INTERFACE I_ENGINE_VALVE EXTENDS I_GENERAL_OBJECT

METHOD M_Close : BOOL
VAR_INPUT
END_VAR
END_METHOD

METHOD M_Open : BOOL
VAR_INPUT
END_VAR
END_METHOD

METHOD M_SetReady : BOOL
VAR_INPUT
END_VAR
END_METHOD

PROPERTY P_Closed : BOOL
GET
END_GET
END_PROPERTY

PROPERTY P_Open : BOOL
GET
END_GET
END_PROPERTY

PROPERTY P_ReadyState : BOOL
GET
END_GET
END_PROPERTY

PROPERTY P_Undefined : BOOL
GET
END_GET
END_PROPERTY

END_INTERFACE

(* stored: Version 1.1.0.1, ProductVersion 3.1.4024.12
   Itf I_ENGINE_VALVE: Id {7e3ceb72-8a0a-4c5a-9e38-262f19a4f12a}
   Method M_Close: Id {2ea4d968-aa32-49e9-92a5-3cfde55592cc}
   Method M_Open: Id {9b168fe1-6505-4f60-9e5c-4242991cd250}
   Method M_SetReady: Id {fdd3cae0-8774-4296-b5ba-55d8bd97d36c}
   Property P_Closed: Id {ff5951e8-0f3a-4262-bf83-1327a1158ec9}
   Get Get: Id {1a09b6d8-8ccb-4b68-ba38-3ee26c837e9f}
   Property P_Open: Id {7cbca0b2-4ae5-4dda-9aed-c8e41f134351}
   Get Get: Id {4f749848-7be1-46fb-bf28-eaa9bc61f912}
   Property P_ReadyState: Id {fb2f8a0d-8c06-4044-a58b-79ae44e1120d}
   Get Get: Id {3daeeb9d-128e-465e-bc11-7525be31476f}
   Property P_Undefined: Id {c32c074c-845b-4d27-9a69-8a835bc82c54}
   Get Get: Id {d85163cf-2547-4c35-a314-1efd1450a0f7} *)
